REGION Network 13 (SCL): COUNT SELECTED BUTTONS
   IF #settings.current.kp8.buttons <> #settings.old.kp8.buttons THEN
       #count := 0;
       FOR #i := 0 TO #buttonCount DO
           #btnSelected := #settings.current.kp8.buttons[#i].select;
           IF #btnSelected THEN
               #count := #count + 1;
           END_IF;
       END_FOR;
       #btnSlctCount := #count;
   END_IF;
END_REGION

REGION Network 14: SELECT ALL BUTTONS
   #tmrSelAllBtn(IN := #settings.current.kp8.assign.act AND NOT #evalSlct AND (#btnSlctCount < #adjBtnCount),   // TON
                 PT := #ptSelectAll);
   IF #tmrSelAllBtn.Q THEN
       "Select All Buttons"(settings := #settings);
       #evalSlct := TRUE;
   END_IF;
END_REGION

REGION Network 15: DESELECT ALL BUTTONS
   #tmrDeslctAllBtn(IN := #settings.current.kp8.assign.act AND NOT #evalSlct AND (#btnSlctCount = #adjBtnCount),   // TON
                    PT := #ptSelectAll);
   IF #tmrDeslctAllBtn.Q THEN
       "Deselect All Buttons"(settings := #settings);
       #evalSlct := TRUE;
   END_IF;
END_REGION

REGION Network 16: RESET EVAL BUTTON SELECTION
   RUNG wire#powerrail
      I_Contact( #settings.current.kp8.assign.act )
      Contact( #settings.old.kp8.assign.act )
      R_Coil( #evalSlct )
   END_RUNG
   // the same network as SCL:
   IF NOT #settings.current.kp8.assign.act AND #settings.old.kp8.assign.act THEN #evalSlct := FALSE; END_IF;
END_REGION

REGION Network 17: ENTRY TIMEOUT
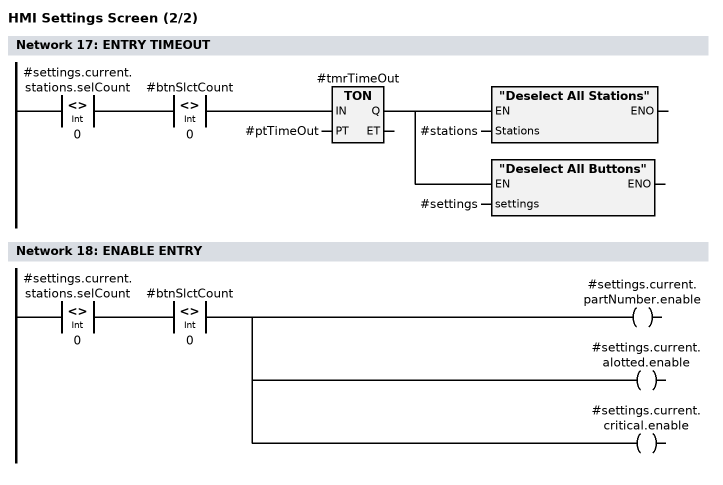
   #tmrTimeOut(IN := (#settings.current.stations.selCount <> 0) AND (#btnSlctCount <> 0), PT := #ptTimeOut);   // TON
   IF #tmrTimeOut.Q THEN
       "Deselect All Stations"(Stations := #stations);
       "Deselect All Buttons"(settings := #settings);
   END_IF;
END_REGION

REGION Network 18: ENABLE ENTRY
   RUNG wire#powerrail
      { S7_Templates := "SrcType := Int" } NE_Contact(in1 := #settings.current.stations.selCount, in2 := 0)
      { S7_Templates := "SrcType := Int" } NE_Contact(in1 := #btnSlctCount, in2 := 0)
      wire#w1
      Coil( #settings.current.partNumber.enable )
   END_RUNG
   RUNG wire#w1
      Coil( #settings.current.alotted.enable )
   END_RUNG
   RUNG wire#w1
      Coil( #settings.current.critical.enable )
   END_RUNG
   // the same network as SCL:
   #settings.current.partNumber.enable := (#settings.current.stations.selCount <> 0) AND (#btnSlctCount <> 0);
   #settings.current.alotted.enable := #settings.current.partNumber.enable;
   #settings.current.critical.enable := #settings.current.partNumber.enable;
END_REGION

REGION Network 19 (SCL): GET BUTTON NUMBER
   IF #btnSlctCount = 1 THEN
       FOR #i := 0 TO #stationCount DO
           #stnSelected := #stations.current[#i].settings.selected;
           IF #stnSelected THEN
               FOR #j := 0 TO #buttonCount DO
                   #btnSelected := #settings.current.kp8.buttons[#j].selState;
                   IF #btnSelected THEN
                       #btnNumber := #j + 1;
                   END_IF;
               END_FOR;
           END_IF;
       END_FOR;
   END_IF;
END_REGION

REGION Network 20 (SCL): DISPLAY PART NUMBER FOR CURRENT BUTTON
   IF #settings.current.viewingStation <> #settings.old.viewingStation THEN
       IF #buttonCount = 1 THEN
           #pSN := #settings.current.viewingStation.number - 1;
           #pBtn := #btnSlctCount - 1;
           #settings.current.partNumber.value := #stations.current[#pSN].partNumbers[#pBtn];
       END_IF;
   END_IF;
END_REGION

REGION Network 21 (SCL): LOAD PART NUMBERS INTO SELECTIONS
   #partNumber := #settings.current.partNumber.value;
   #oldPN := #settings.old.partNumber.value;
   #newEntry := FALSE;
   IF #partNumber <> #oldPN THEN
       #newEntry := TRUE;
   END_IF;
   IF #newEntry THEN
       #newEntry := FALSE;
       FOR #i := 0 TO #constants.stationCount DO
           #stnSelected := #stations.current[#i].settings.selected;
           IF #stnSelected THEN
               FOR #j := 0 TO #constants.buttonCount DO
                   #btnSelected := #settings.current.kp8.buttons[#j].selState;
                   IF #btnSelected THEN
                       #stations.current[#i].partNumbers[#j] := #partNumber;
                   END_IF;
               END_FOR;
           END_IF;
       END_FOR;
   END_IF;
END_REGION

REGION Network 22 (SCL): LOAD TIMER VALUES INTO SELECTIONS
   #currentBtn := #settings.current.alotted.setTimer;
   #oldBtn := #settings.old.alotted.setTimer;
   IF #currentBtn AND NOT #oldBtn THEN
       #timerWString := #settings.current.alotted.value;
       FOR #i := 0 TO #constants.stationCount - 1 DO
           #stnSelected := #stations.current[#i].settings.selected;
           IF #stnSelected THEN
               FOR #j := 0 TO #constants.buttonCount - 1 DO
                   #btnSelected := #settings.current.kp8.buttons[#j].select;
                   IF #btnSelected THEN
                       #stations.current[#i].presetTime.allotted[#j] := "WString Timer to Real"(#timerWString);
                   END_IF;
               END_FOR;
           END_IF;
       END_FOR;
   END_IF;
END_REGION

REGION Network 23 (SCL): LOAD CRITICAL TIME VALUES INTO SELECTIONS
   #currentBtn := #settings.current.critical.setTimer;
   #oldBtn := #settings.old.critical.setTimer;

   IF #currentBtn AND NOT #oldBtn THEN
       #timerWString := #settings.current.alotted.value;
       FOR #i := 0 TO #constants.stationCount - 1 DO
           #stnSelected := #stations.current[#i].settings.selected;
           IF #stnSelected THEN
               FOR #j := 0 TO #constants.buttonCount - 1 DO
                   #btnSelected := #settings.current.kp8.buttons[#j].select;
                   IF #btnSelected THEN
                       #stations.current[#i].presetTime.critical[#j] := "WString Timer to Real"(#timerWString);
                   END_IF;
               END_FOR;
           END_IF;
       END_FOR;
   END_IF;
END_REGION

REGION Network 24 (SCL): UPDATE CURRENT STATION VIEW PORT
   #currentBtn := #settings.current.partNumber.enter OR
                   #settings.current.alotted.setTimer OR
                   #settings.current.critical.setTimer;
   #oldBtn := #settings.old.partNumber.enter OR
                   #settings.old.alotted.setTimer OR
                   #settings.old.critical.setTimer;
   #stnNumber := #settings.current.viewingStation.number;
   #oldStnNumber := #settings.old.viewingStation.number;
   IF (#currentBtn AND NOT #oldBtn) OR
       (#stnNumber <> #oldStnNumber) THEN
       #pSN := #stnNumber - 1;
           // station number: see network 5 & 6
           // line value
           #settings.current.viewingStation.lineValue := #stations.current[#pSN].line;
           // drop zone
           #settings.current.viewingStation.dzValue := #stations.current[#pSN].dropZone;
           // loop through buttons
           FOR #i := 0 TO #constants.buttonCount - 1 DO
               // part number
               #partNumber := #stations.current[#pSN].partNumbers[#i];
               #settings.current.viewingStation.btns[#i].partNumber := #partNumber;
               // allotted time
               #timerWString := "Real to WString Timer"(#stations.current[#pSN].presetTime.allotted[#i]);
               #settings.current.viewingStation.btns[#i].alloted := #timerWString;
               // critical time
               #timerWString := "Real to WString Timer"(#stations.current[#pSN].presetTime.critical[#i]);
               #settings.current.viewingStation.btns[#i].critical := #timerWString;
           END_FOR;
   END_IF;
END_REGION
END_FUNCTION_BLOCK

FUNCTION_BLOCK "Collapse Table"   // FB15, SCL
{ S7_Optimized_Access := 'TRUE' }
VERSION : 0.1
   VAR_INPUT
      constants : "Constants";
   END_VAR
   VAR_IN_OUT
      requests : "Part Request Data";
   END_VAR
   VAR
      tableBox : "Part Request Data";
   END_VAR
   VAR_TEMP
      blankRow : "Table Row";
      collapseReq : Bool;
      i : Int;
      maxRows : Int;
      pCollapse : Int;
   END_VAR
BEGIN
   REGION "COPY TO LOCAL"
       #maxRows := #constants.partReqRows - 1;
   END_REGION

   REGION "REMOVE EMPTY ROWS"
       FOR #i := 0 TO #maxRows DO

           REGION "ROW IS NOT EMPTY"
               IF #requests.row[#i].address <> 0 THEN

                   REGION "MOVE TO TEMP TABLE"
                       #tableBox.row[#pCollapse] := #requests.row[#i];
                   END_REGION

                   REGION "POINTERS AND FLAGS"
                       #pCollapse := #pCollapse + 1;
                       #collapseReq := TRUE;
                   END_REGION

               END_IF;
           END_REGION

       END_FOR;
   END_REGION

   REGION "COLLAPSE TABLE"
       IF #collapseReq THEN

           REGION "TURN OFF THE LIGHTS"
               #collapseReq := FALSE;
           END_REGION

           REGION "COPY TEMP TO PERMANENT"
               #requests := #tableBox;
           END_REGION

           REGION "CLEAR VALUES FROM TEMP TABLE"
               FOR #i := 0 TO #maxRows DO
                   #tableBox.row[#i] := #blankRow;
               END_FOR;
           END_REGION
       END_IF;

   END_REGION
END_FUNCTION_BLOCK

FUNCTION_BLOCK "HMI Populate Part Call"   // FB16, SCL
{ S7_Optimized_Access := 'TRUE' }
VERSION : 0.1
   VAR_INPUT
      constants : "Constants";
      requests : "Part Request Data";
   END_VAR
   VAR_IN_OUT
      partCall : "Part Call Screen";
   END_VAR
   VAR
      pDisplay : Int;
   END_VAR
   VAR_TEMP
      firstRow : Int;
      i : Int;
      lastRow : Int;
      maxRows : Int;
      pRow : Int;
      visibleRows : Int;
      thisRow : Int;
   END_VAR
BEGIN
   #visibleRows := #constants.hmiRowCount - 1;
   #maxRows := #constants.partReqRows - 1;
   #firstRow := 0;
   #lastRow := #firstRow + #visibleRows;

   FOR #i := 0 TO #visibleRows DO
       #partCall.current[#i] := #requests.row[#i];
   END_FOR;
END_FUNCTION_BLOCK

FUNCTION_BLOCK "KP8 Driver"   // FB101, SCL
{ S7_Optimized_Access := 'FALSE' }
VERSION : 0.1
   VAR_INPUT
      btnIn : Byte;   // byte that contains input data from kp8 buttons
      hardInit : Bool;   // initializes function. can be used for reset
      softInit : Bool;
      btn0Activate : Bool;   // true for on, false for off
      btn0Mode : Bool;   // true for maintained, false for momentary
      btn0Group : Int;
      btn0Flash : Bool;
      btn0ColorOn1 : String[10];   // enter: red OR green OR blue OR yellow OR white OR off
      btn0ColorOn2 : String[10];
      btn0ColorOff : String[10];   // enter: red OR green OR blue OR yellow OR white OR off
      btn1Activate : Bool;   // true for on, false for off
      btn1Mode : Bool;   // true for maintained, false for momentary
      btn1Group : Int;
      btn1Flash : Bool;
      btn1ColorOn1 : String[10];   // enter: red OR green OR blue OR yellow OR white OR off
      btn1ColorOn2 : String[10];
      btn1ColorOff : String[10];   // enter: red OR green OR blue OR yellow OR white OR off
      btn2Activate : Bool;   // true for on, false for off
      btn2Mode : Bool;   // true for maintained, false for momentary
      btn2Group : Int;
      btn2Flash : Bool;
      btn2ColorOn1 : String[10] := '';   // enter: red OR green OR blue OR yellow OR white OR off
      btn2ColorOn2 : String[10];
      btn2ColorOff : String[10];   // enter: red OR green OR blue OR yellow OR white OR off
      btn3Activate : Bool;   // true for on, false for off
      btn3Mode : Bool;   // true for maintained, false for momentary
      btn3Group : Int;
      btn3Flash : Bool;
      btn3ColorOn1 : String[10];   // enter: red OR green OR blue OR yellow OR white OR off
      btn3ColorOn2 : String[10];
      btn3ColorOff : String[10];   // enter: red OR green OR blue OR yellow OR white OR off
      btn4Activate : Bool;   // true for on, false for off
      btn4Mode : Bool;   // true for maintained, false for momentary
      btn4Group : Int;
      btn4Flash : Bool;
      btn4ColorOn1 : String[10];   // enter: red OR green OR blue OR yellow OR white OR off
      btn4ColorOn2 : String[10];
      btn4ColorOff : String[10];   // enter: red OR green OR blue OR yellow OR white OR off
      btn5Activate : Bool;   // true for on, false for off
      btn5Mode : Bool;   // true for maintained, false for momentary
      btn5Group : Int;
      btn5Flash : Bool;
      btn5ColorOn1 : String[10];   // enter: red OR green OR blue OR yellow OR white OR off
      btn5ColorOn2 : String[10];
      btn5ColorOff : String[10];   // enter: red OR green OR blue OR yellow OR white OR off
      btn6Activate : Bool;   // true for on, false for off
      btn6Mode : Bool;   // true for maintained, false for momentary
      btn6Group : Int;
      btn6Flash : Bool;
      btn6ColorOn1 : String[10];   // enter: red OR green OR blue OR yellow OR white OR off
      btn6ColorOn2 : String[10];
      btn6ColorOff : String[10];   // enter: red OR green OR blue OR yellow OR white OR off
      btn7Activate : Bool;   // true for on, false for off
      btn7Mode : Bool;   // true for maintained, false for momentary
      btn7Group : Int;
      btn7Flash : Bool;
      btn7ColorOn1 : String[10];   // enter: red OR green OR blue OR yellow OR white OR off
      btn7ColorOn2 : String[10];
      btn7ColorOff : String[10];   // enter: red OR green OR blue OR yellow OR white OR off
   END_VAR
   VAR_OUTPUT
      btnStatesOut : Array[0..7] of Bool;   // the output array represents the state of button presses
      btnColorsOut : DWord;
   END_VAR
   VAR
      mask : Byte;
      btnInInt : Byte;
      btnEval : Byte;
      i1 : Int;
      i2 : Int;
      btnInArrayNew : Array[0..7] of Bool;
      btnInArrayOld : Array[0..7] of Bool;
      btnStateArrayInt : Array[0..7] of Bool;
      btnActivateInt : Array[0..7] of Bool;
      btnModeInt : Array[0..7] of Bool;
      btnFlashInt : Array[0..7] of Bool;
      btnGroup : Array[0..7] of Int;
      btnClrMskOn1Int : Array[0..7] of DWord;
      btnClrMskOn2Int : Array[0..7] of DWord;
      btnClrMskOffInt : Array[0..7] of DWord;
      btnClrOn1Int : Array[0..7] of String[10];
      btnClrOn2Int : Array[0..7] of String[10];
      btnClrOffInt : Array[0..7] of String[10];
   END_VAR
   VAR CONSTANT
      btnMskRed : DWord := dw#16#0100_0000;
      btnMskGreen : DWord := dw#16#0001_0000;
      btnMskBlue : DWord := dw#16#000_0100;
      btnMskYellow : DWord := dw#16#0101_0000;
      btnMskWhite : DWord := dw#16#0101_0100;
      btnMskBlack : DWord := dw#16#FEFE_FEFF;
      initBtnColors : DWord := dw#16#0000_0000;
   END_VAR
BEGIN
   REGION "ALL INITS"
       IF #hardInit OR #softInit THEN

           REGION "CLEAR OUTPUT COLORS"
               #btnColorsOut := #initBtnColors;
           END_REGION

           REGION "TRANSFER PARAMETERS TO INTERNAL ARRAYS"

               REGION "BUTTON 0"
                   #btnActivateInt[0] := #btn0Activate;
                   #btnModeInt[0] := #btn0Mode;
                   #btnGroup[0] := #btn0Group;
                   #btnClrOn1Int[0] := #btn0ColorOn1;
                   #btnClrOn2Int[0] := #btn0ColorOn2;
                   #btnClrOffInt[0] := #btn0ColorOff;
               END_REGION

               REGION "BUTTON 1"
                   #btnActivateInt[1] := #btn1Activate;
                   #btnModeInt[1] := #btn1Mode;
                   #btnGroup[1] := #btn1Group;
                   #btnClrOn1Int[1] := #btn1ColorOn1;
                   #btnClrOn2Int[1] := #btn1ColorOn2;
                   #btnClrOffInt[1] := #btn1ColorOff;
               END_REGION

               REGION "BUTTON 2"
                   #btnActivateInt[2] := #btn2Activate;
                   #btnModeInt[2] := #btn2Mode;
                   #btnGroup[2] := #btn2Group;
                   #btnClrOn1Int[2] := #btn2ColorOn1;
                   #btnClrOn2Int[2] := #btn2ColorOn2;
                   #btnClrOffInt[2] := #btn2ColorOff;
               END_REGION

               REGION "BUTTON 3"
                   #btnActivateInt[3] := #btn3Activate;
                   #btnModeInt[3] := #btn3Mode;
                   #btnGroup[3] := #btn3Group;
                   #btnClrOn1Int[3] := #btn3ColorOn1;
                   #btnClrOn2Int[3] := #btn3ColorOn2;
                   #btnClrOffInt[3] := #btn3ColorOff;
               END_REGION

               REGION "BUTTON 4"
                   #btnActivateInt[4] := #btn4Activate;
                   #btnModeInt[4] := #btn4Mode;
                   #btnGroup[4] := #btn4Group;
                   #btnClrOn1Int[4] := #btn4ColorOn1;
                   #btnClrOn2Int[4] := #btn4ColorOn2;
                   #btnClrOffInt[4] := #btn4ColorOff;
               END_REGION

               REGION "BUTTON 5"
                   #btnActivateInt[5] := #btn5Activate;
                   #btnModeInt[5] := #btn5Mode;
                   #btnGroup[5] := #btn5Group;
                   #btnClrOn1Int[5] := #btn5ColorOn1;
                   #btnClrOn2Int[5] := #btn5ColorOn2;
                   #btnClrOffInt[5] := #btn5ColorOff;
               END_REGION

               REGION "BUTTON 6"
                   #btnActivateInt[6] := #btn6Activate;
                   #btnModeInt[6] := #btn6Mode;
                   #btnGroup[6] := #btn6Group;
                   #btnClrOn1Int[6] := #btn6ColorOn1;
                   #btnClrOn2Int[6] := #btn6ColorOn2;
                   #btnClrOffInt[6] := #btn6ColorOff;
               END_REGION

               REGION "BUTTON 7"
                   #btnActivateInt[7] := #btn7Activate;
                   #btnModeInt[7] := #btn7Mode;
                   #btnGroup[7] := #btn7Group;
                   #btnClrOn1Int[7] := #btn7ColorOn1;
                   #btnClrOn2Int[7] := #btn7ColorOn2;
                   #btnClrOffInt[7] := #btn7ColorOff;
               END_REGION

           END_REGION

           REGION "RECOLOR BUTTON MASKS"
               FOR #i1 := 0 TO 7 DO

                   REGION "ON COLOR 1"
                       IF (#btnClrOn1Int[#i1] = 'red') THEN
                           #btnClrMskOn1Int[#i1] := SHL(IN := #btnMskRed, N := #i1);
                       ELSIF (#btnClrOn1Int[#i1] = 'green') THEN
                           #btnClrMskOn1Int[#i1] := SHL(IN := #btnMskGreen, N := #i1);
                       ELSIF (#btnClrOn1Int[#i1] = 'blue') THEN
                           #btnClrMskOn1Int[#i1] := SHL(IN := #btnMskBlue, N := #i1);
                       ELSIF (#btnClrOn1Int[#i1] = 'yellow') THEN
                           #btnClrMskOn1Int[#i1] := SHL(IN := #btnMskYellow, N := #i1);
                       ELSIF (#btnClrOn1Int[#i1] = 'white') THEN
                           #btnClrMskOn1Int[#i1] := SHL(IN := #btnMskWhite, N := #i1);
                       ELSIF (#btnClrOn1Int[#i1] = 'off') THEN
                           #btnClrMskOn1Int[#i1] := 0;
                       END_IF;
                   END_REGION

                   REGION "ON COLOR 2"
                       IF (#btnClrOn2Int[#i1] = 'red') THEN
                           #btnClrMskOn2Int[#i1] := SHL(IN := #btnMskRed, N := #i1);
                       ELSIF (#btnClrOn2Int[#i1] = 'green') THEN
                           #btnClrMskOn2Int[#i1] := SHL(IN := #btnMskGreen, N := #i1);
                       ELSIF (#btnClrOn2Int[#i1] = 'blue') THEN
                           #btnClrMskOn2Int[#i1] := SHL(IN := #btnMskBlue, N := #i1);
                       ELSIF (#btnClrOn2Int[#i1] = 'yellow') THEN
                           #btnClrMskOn2Int[#i1] := SHL(IN := #btnMskYellow, N := #i1);
                       ELSIF (#btnClrOn2Int[#i1] = 'white') THEN
                           #btnClrMskOn2Int[#i1] := SHL(IN := #btnMskWhite, N := #i1);
                       ELSIF (#btnClrOn2Int[#i1] = 'off') THEN
                           #btnClrMskOn2Int[#i1] := 0;
                       END_IF;
                   END_REGION

                   REGION "OFF COLOR"
                       IF (#btnClrOffInt[#i1] = 'red') THEN
                           #btnClrMskOffInt[#i1] := SHL(IN := #btnMskRed, N := #i1);
                       ELSIF (#btnClrOffInt[#i1] = 'green') THEN
                           #btnClrMskOffInt[#i1] := SHL(IN := #btnMskGreen, N := #i1);
                       ELSIF (#btnClrOffInt[#i1] = 'blue') THEN
                           #btnClrMskOffInt[#i1] := SHL(IN := #btnMskBlue, N := #i1);
                       ELSIF (#btnClrOffInt[#i1] = 'yellow') THEN
                           #btnClrMskOffInt[#i1] := SHL(IN := #btnMskYellow, N := #i1);
                       ELSIF (#btnClrOffInt[#i1] = 'white') THEN
                           #btnClrMskOffInt[#i1] := SHL(IN := #btnMskWhite, N := #i1);
                       ELSIF (#btnClrOffInt[#i1] = 'off') THEN
                           #btnClrMskOffInt[#i1] := 0;
                       END_IF;
                   END_REGION

               END_FOR;
           END_REGION

       END_IF;
   END_REGION

   REGION "HART INIT"
       IF #hardInit THEN
           FOR #i1 := 0 TO 7 DO
               #btnStateArrayInt[#i1] := FALSE;
           END_FOR;
       END_IF;
   END_REGION


   REGION "TRANFER PARAMETERS TO ARRAYS"
       // raw pb data
       #btnInInt := #btnIn;
       // flashing modes
       #btnFlashInt[0] := #btn0Flash;
       #btnFlashInt[1] := #btn1Flash;
       #btnFlashInt[2] := #btn2Flash;
       #btnFlashInt[3] := #btn3Flash;
       #btnFlashInt[4] := #btn4Flash;
       #btnFlashInt[5] := #btn5Flash;
       #btnFlashInt[6] := #btn6Flash;
       #btnFlashInt[7] := #btn7Flash;
   END_REGION

   REGION "EVALUATE BUTTONS"
       FOR #i1 := 0 TO 7 DO

           REGION "TRANSFER BUTTON PRESSES TO ARRAY"
               #btnEval := SHR(IN := #btnInInt, N := #i1);
               #btnInArrayNew[#i1] := #btnEval.%X0;
               #btnEval := b#16#0;
           END_REGION

           REGION "SET BUTTON STATE"

               REGION "BUTTON ACTIVE"
                   IF #btnActivateInt[#i1] THEN

                       REGION "MAINTAINED"
                           IF #btnModeInt[#i1] THEN

                               REGION "RISING EDGE OF PRESS"
                                   IF #btnInArrayNew[#i1] AND NOT #btnInArrayOld[#i1] THEN

                                       REGION "CHECK FOR GROUP MEMBERSHIP"
                                           FOR #i2 := 0 TO 7 DO

                                               REGION "NOT IN NULL GROUP"
                                                   IF (#btnGroup[#i2] <> 0) THEN

                                                       REGION "SKIP SELF"
                                                           IF (#i2 <> #i1) THEN

                                                               REGION "GROUPS MATCH"
                                                                   IF #btnGroup[#i1] = #btnGroup[#i2] THEN
                                                                       REGION "DEACTIVATE OTHER GROUP MEMBERS"
                                                                           #btnStateArrayInt[#i2] := FALSE;
                                                                       END_REGION

                                                                   END_IF;
                                                               END_REGION

                                                           END_IF;
                                                       END_REGION

                                                   END_IF;
                                               END_REGION

                                           END_FOR;
                                       END_REGION

                                       REGION "TOGGLE STATE"
                                           #btnStateArrayInt[#i1] := NOT #btnStateArrayInt[#i1];
                                       END_REGION

                                   END_IF;
                               END_REGION

                           END_IF;
                       END_REGION

                       REGION "MOMENTARY"
                           IF NOT #btnModeInt[#i1] THEN
                               #btnStateArrayInt[#i1] := #btnInArrayNew[#i1];
                           END_IF;
                       END_REGION

                   END_IF;
               END_REGION

               REGION "BUTTON INACTIVE"
                   IF NOT #btnActivateInt[#i1] THEN
                       #btnStateArrayInt[#i1] := FALSE;
                   END_IF;
               END_REGION

           END_REGION

           REGION "ANIMATE BUTTONS"

               REGION "BUTTON ON FLASH BIT OFF"
                   IF #btnStateArrayInt[#i1] AND NOT #btnFlashInt[#i1] THEN
                       #btnColorsOut := #btnColorsOut AND ROL(IN := #btnMskBlack, N := #i1);
                       #btnColorsOut := #btnColorsOut OR #btnClrMskOn1Int[#i1];
                   END_IF;
               END_REGION

               REGION "BUTTON ON FLASH BIT ON"
                   IF #btnStateArrayInt[#i1] AND #btnFlashInt[#i1] THEN
                       #btnColorsOut := #btnColorsOut AND ROL(IN := #btnMskBlack, N := #i1);
                       #btnColorsOut := #btnColorsOut OR #btnClrMskOn2Int[#i1];
                   END_IF;
               END_REGION

               REGION "BUTTON OFF"
                   IF NOT #btnStateArrayInt[#i1] THEN
                       #btnColorsOut := #btnColorsOut AND ROL(IN := #btnMskBlack, N := #i1);
                       #btnColorsOut := #btnColorsOut OR #btnClrMskOffInt[#i1];
                   END_IF;
               END_REGION

           END_REGION

       END_FOR;
   END_REGION

   REGION "CHANGE DETECTION"
       #btnInArrayOld := #btnInArrayNew;
   END_REGION

   REGION "OUTPUT"
       #btnStatesOut := #btnStateArrayInt;
   END_REGION
END_FUNCTION_BLOCK

FUNCTION "Physical to Global" : Void   // FC1, LAD
{ S7_Optimized_Access := 'TRUE' }
VERSION : 0.1
   VAR_INPUT
      constants : "Constants";
   END_VAR
   VAR_IN_OUT
      stations : "Stations";
   END_VAR
   VAR_TEMP
      i : Int;
      kp8In : DWord;
      stnCount : Int;
   END_VAR
   VAR CONSTANT
      "VOLVO 16 1" : Int := 0;
      "VOLVO 16 2" : Int := 1;
      "VOLVO 16 3" : Int := 2;
      "VOLVO 16 4" : Int := 3;
      "VOLVO 16 5" : Int := 4;
      "VOLVO 16 6" : Int := 5;
      "VOLVO 16 7" : Int := 6;
      "VOLVO 16 8" : Int := 7;
      "VOLVO 16 9" : Int := 8;
      "VOLVO 16 10" : Int := 9;
      "VOLVO 16 11" : Int := 10;
      "CHM 1" : Int := 11;
      "CHM 2" : Int := 12;
      "CHM 3" : Int := 13;
      "CHM 4" : Int := 14;
      "CDO 1" : Int := 15;
      "CDO 2" : Int := 16;
      "CDO 3" : Int := 17;
      "BFL 1" : Int := 18;
      "BFL 2" : Int := 19;
      "BFL 3" : Int := 20;
      "LGS 1" : Int := 21;
      "LGS 2" : Int := 22;
   END_VAR
BEGIN

REGION Network 1
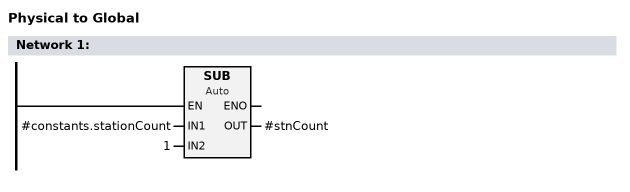
   RUNG wire#powerrail
      Sub(in1 := #constants.stationCount, in2 := 1, out => #stnCount)
   END_RUNG
   // the same network as SCL:
   #stnCount := #constants.stationCount - 1;
END_REGION

REGION Network 2 (SCL): MAIN LOOP
   FOR #i := 0 TO #stnCount DO

       CASE #i OF
           #"VOLVO 16 1":
               #kp8In := "VOLVO 16 1 KP8 In";
           #"VOLVO 16 2":
               #kp8In := "VOLVO 16 2 KP8 In";
           #"VOLVO 16 3":
               #kp8In := "VOLVO 16 3 KP8 In";
           #"VOLVO 16 4":
               #kp8In := "VOLVO 16 4 KP8 In";
           #"VOLVO 16 5":
               #kp8In := "VOLVO 16 5 KP8 In";
           #"VOLVO 16 6":
               #kp8In := "VOLVO 16 6 KP8 In";
           #"VOLVO 16 7":
               #kp8In := "VOLVO 16 7 KP8 In";
           #"VOLVO 16 8":
               #kp8In := "VOLVO 16 8 KP8 In";
           #"VOLVO 16 9":
               #kp8In := "VOLVO 16 9 KP8 In";
           #"VOLVO 16 10":
               #kp8In := "VOLVO 16 10 KP8 In";
           #"VOLVO 16 11":
               #kp8In := "VOLVO 16 11 KP8 In";
           #"CHM 1":
               #kp8In := "CHM 1 KP8 In";
           #"CHM 2":
               #kp8In := "CHM 2 KP8 In";
           #"CHM 3":
               #kp8In := "CHM 3 KP8 In";
           #"CHM 4":
               #kp8In := "CHM 4 KP8 In";
           #"CDO 1":
               #kp8In := "CDO 1 KP8 In";
           #"CDO 2":
               #kp8In := "CDO 2 KP8 In";
           #"CDO 3":
               #kp8In := "CDO 3 KP8 In";
           #"BFL 1":
               #kp8In := "BFL 1 KP8 In";
           #"BFL 2":
               #kp8In := "BFL 2 KP8 In";
           #"BFL 3":
               #kp8In := "BFL 3 KP8 In";
           #"LGS 1":
               #kp8In := "LGS 1 KP8 In";
           #"LGS 2":
               #kp8In := "LGS 2 KP8 In";

       END_CASE;

       #stations.current[#i].kp8In := #kp8In.%B3;

   END_FOR;
END_REGION
END_FUNCTION

FUNCTION "Time to WString" : WString   // FC2, SCL
{ S7_Optimized_Access := 'TRUE' }
VERSION : 0.1
   VAR_INPUT
      "Time" : Time;
   END_VAR
   VAR_TEMP
      "Time as DInt" : DInt;
      "Hours 10s Place" : DInt;
      "Hours 1s Place" : DInt;
      "Minutes 10s Place" : DInt;
      "Minutes 1s Place" : DInt;
      "Seconds 10s Place" : DInt;
      "Seconds 1s Place" : DInt;
      "Time Elements" : Array[0..4] of WString;
      Length : Int;
      "String Box" : WString;
      "DInt Box" : DInt;
   END_VAR
   VAR CONSTANT
      "Milliseconds per 10 Hours" : DInt := 36000000;
      "Milliseconds per Hour" : DInt := 3600000;
      "Milliseconds per 10 Minutes" : DInt := 600000;
      "Milliseconds per Minute" : DInt := 60000;
      "Milliseconds per 10 Seconds" : DInt := 10000;
      "Milliseconds per Second" : DInt := 1000;
   END_VAR
BEGIN
   REGION GET INPUT
       #"Time as DInt" := #Time;
   END_REGION

   REGION CONVERT TIME INTO INDIVIDUAL PLACE VALUES
       #"Minutes 10s Place" := #"Time as DInt" / #"Milliseconds per 10 Minutes";
       #"Minutes 1s Place" := (#"Time as DInt" / #"Milliseconds per Minute") MOD 10;
       #"Seconds 10s Place" := (#"Time as DInt" MOD #"Milliseconds per Minute") / #"Milliseconds per 10 Seconds";
       #"Seconds 1s Place" := (#"Time as DInt" / #"Milliseconds per Second") MOD 10;
   END_REGION

   REGION "ADD SIGN"
       #"Time Elements"[0] := wstring#'';
       IF #"Minutes 10s Place" < 0 OR
           #"Minutes 1s Place" < 0 OR
           #"Seconds 10s Place" < 0 OR
           #"Seconds 1s Place" < 0 THEN
            #"Time Elements"[0] := wstring#'-';
       END_IF;
   END_REGION

   REGION CONVERT PLACE VALUES INTO COMPONENT STRINGS
       // MINUTES
       #"DInt Box" := #"Minutes 10s Place" * 10 + #"Minutes 1s Place";
       #"String Box" := DINT_TO_WSTRING(IN := #"DInt Box");
       #"String Box" := "Strip Sign"("WString":=#"String Box");
       #"String Box" := "Add Leading"("Leading Character" := WCHAR#'0',
                                      "Desired Length" := 2,
                                      "String" := #"String Box");
       #"Time Elements"[1] := #"String Box";
       // COLON
       #"Time Elements"[2] := WSTRING#':';
       // SECONDS
       #"DInt Box" := #"Seconds 10s Place" * 10 + #"Seconds 1s Place";
       #"String Box" := DINT_TO_WSTRING(IN := #"DInt Box");
       #"String Box" := "Strip Sign"("WString":=#"String Box");
       #"String Box" := "Add Leading"("Leading Character" := WCHAR#'0',
                                      "Desired Length" := 2,
                                      "String" := #"String Box");
       #"Time Elements"[3] := #"String Box";
   END_REGION


   REGION RETURN VALUE
       #"Time to WString" := CONCAT_WSTRING(IN1 := #"Time Elements"[0],
                                            IN2 := #"Time Elements"[1],
                                            IN3 := #"Time Elements"[2],
                                            IN4 := #"Time Elements"[3]);
   END_REGION
END_FUNCTION

FUNCTION "Strip Sign" : WString   // FC3, SCL
{ S7_Optimized_Access := 'TRUE' }
VERSION : 0.1
   VAR_INPUT
      WString : WString;
   END_VAR
   VAR_TEMP
      Length : Int;
      "String Box" : WString;
      "Test Character" : WString;
   END_VAR
   VAR CONSTANT
      "+" : WChar := WCHAR#'+';
      "-" : WChar := WCHAR#'-';
   END_VAR
BEGIN
   #"String Box" := #WString;
   #"Test Character" := LEFT_WSTRING(IN := #"String Box",
                                     L := 1);
   IF #"Test Character" = #"+" OR #"Test Character" = #"-" THEN
       #Length := LEN(#"String Box");
       #"String Box" := RIGHT_WSTRING(IN := #"String Box", L := #Length - 1);

   END_IF;
   #"Strip Sign" := #"String Box";
END_FUNCTION

FUNCTION "Add Leading" : WString   // FC4, SCL
{ S7_Optimized_Access := 'TRUE' }
VERSION : 0.1
   VAR_INPUT
      "Leading Character" : WChar;
      "Desired Length" : USInt;
      "String" : WString;
   END_VAR
   VAR_TEMP
      Length : Int;
      "String Box" : WString;
      Constant : WString;
   END_VAR
BEGIN
   #"String Box" := #String;
   #Length := LEN(#"String Box");

   WHILE #Length < #"Desired Length" DO
       #"String Box" := CONCAT_WSTRING(IN1 := #"Leading Character",
                                       IN2 := #"String Box");
       #Length := LEN(#"String Box");
   END_WHILE;

   #"Add Leading" := #"String Box";
END_FUNCTION

FUNCTION "Global to Physical" : Void   // FC5, LAD
{ S7_Optimized_Access := 'TRUE' }
VERSION : 0.1
   VAR_INPUT
      constants : "Constants";
   END_VAR
   VAR_IN_OUT
      stations : "Stations";
   END_VAR
   VAR_TEMP
      i : Int;
      j : Int;
      IO : DWord;
      "KP8 In" : DWord;
      "KP8 Out" : DWord;
      Card : Int;
      stnCount : Int;
   END_VAR
   VAR CONSTANT
      "VOLVO 16 1" : Int := 0;
      "VOLVO 16 2" : Int := 1;
      "VOLVO 16 3" : Int := 2;
      "VOLVO 16 4" : Int := 3;
      "VOLVO 16 5" : Int := 4;
      "VOLVO 16 6" : Int := 5;
      "VOLVO 16 7" : Int := 6;
      "VOLVO 16 8" : Int := 7;
      "VOLVO 16 9" : Int := 8;
      "VOLVO 16 10" : Int := 9;
      "VOLVO 16 11" : Int := 10;
      "CHM 1" : Int := 11;
      "CHM 2" : Int := 12;
      "CHM 3" : Int := 13;
      "CHM 4" : Int := 14;
      "CDO 1" : Int := 15;
      "CDO 2" : Int := 16;
      "CDO 3" : Int := 17;
      "BFL 1" : Int := 18;
      "BFL 2" : Int := 19;
      "BFL 3" : Int := 20;
      "LGS 1" : Int := 21;
      "LGS 2" : Int := 22;
   END_VAR
BEGIN

REGION Network 1: ARRAY LIMIT FOR STATION COUNT
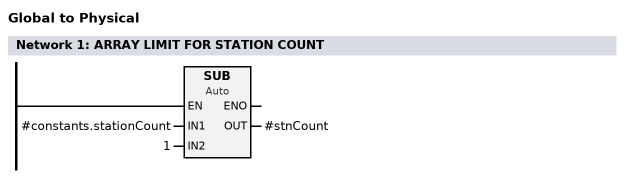
   RUNG wire#powerrail
      Sub(in1 := #constants.stationCount, in2 := 1, out => #stnCount)
   END_RUNG
   // the same network as SCL:
   #stnCount := #constants.stationCount - 1;
END_REGION

REGION Network 2 (SCL): MAIN LOOP
   FOR #i := 0 TO #stnCount DO

       #IO := #stations.current[#i].stackLightOut;
       #"KP8 Out" := #stations.current[#i].kp8Out;

       CASE #i OF
           #"VOLVO 16 1":
               "VOLVO 16 1 IO" := #IO;
               "VOLVO 16 1 KP8 Out" := #"KP8 Out";
           #"VOLVO 16 2":
               "VOLVO 16 2 IO" := #IO;
               "VOLVO 16 2 KP8 Out" := #"KP8 Out";
           #"VOLVO 16 3":
               "VOLVO 16 3 IO" := #IO;
               "VOLVO 16 3 KP8 Out" := #"KP8 Out";
           #"VOLVO 16 4":
               "VOLVO 16 4 IO" := #IO;
               "VOLVO 16 4 KP8 Out" := #"KP8 Out";
           #"VOLVO 16 5":
               "VOLVO 16 5 IO" := #IO;
               "VOLVO 16 5 KP8 Out" := #"KP8 Out";
           #"VOLVO 16 6":
               "VOLVO 16 6 IO" := #IO;
               "VOLVO 16 6 KP8 Out" := #"KP8 Out";
           #"VOLVO 16 7":
               "VOLVO 16 7 IO" := #IO;
               "VOLVO 16 7 KP8 Out" := #"KP8 Out";
           #"VOLVO 16 8":
               "VOLVO 16 8 IO" := #IO;
               "VOLVO 16 8 KP8 Out" := #"KP8 Out";
           #"VOLVO 16 9":
               "VOLVO 16 9 IO" := #IO;
               "VOLVO 16 9 KP8 Out" := #"KP8 Out";
           #"VOLVO 16 10":
               "VOLVO 16 10 IO" := #IO;
               "VOLVO 16 10 KP8 Out" := #"KP8 Out";
           #"VOLVO 16 11":
               "VOLVO 16 11 IO" := #IO;
               "VOLVO 16 11 KP8 Out" := #"KP8 Out";
           #"CHM 1":
               "CHM 1 IO" := #IO;
               "CHM 1 KP8 Out" := #"KP8 Out";
           #"CHM 2":
               "CHM 2 IO" := #IO;
               "CHM 2 KP8 Out" := #"KP8 Out";
           #"CHM 3":
               "CHM 3 IO" := #IO;
               "CHM 3 KP8 Out" := #"KP8 Out";
           #"CHM 4":
               "CHM 4 IO" := #IO;
               "CHM 4 KP8 Out" := #"KP8 Out";
           #"CDO 1":
               "CDO 1 IO" := #IO;
               "CDO 1 KP8 Out" := #"KP8 Out";
           #"CDO 2":
               "CDO 2 IO" := #IO;
               "CDO 2 KP8 Out" := #"KP8 Out";
           #"CDO 3":
               "CDO 3 IO" := #IO;
               "CDO 3 KP8 Out" := #"KP8 Out";
           #"BFL 1":
               "BFL 1 IO" := #IO;
               "BFL 1 KP8 Out" := #"KP8 Out";
           #"BFL 2":
               "BFL 2 IO" := #IO;
               "BFL 2 KP8 Out" := #"KP8 Out";
           #"BFL 3":
               "BFL 3 IO" := #IO;
               "BFL 3 KP8 Out" := #"KP8 Out";
           #"LGS 1":
               "LGS 1 IO" := #IO;
               "LGS 1 KP8 Out" := #"KP8 Out";
           #"LGS 2":
               "LGS 2 IO" := #IO;
               "LGS 2 KP8 Out" := #"KP8 Out";

       END_CASE;

   END_FOR;
END_REGION
END_FUNCTION

FUNCTION "Select All Stations" : Void   // FC6, SCL
{ S7_Optimized_Access := 'TRUE' }
VERSION : 0.1
   VAR_IN_OUT
      stations : "Stations";
   END_VAR
   VAR_TEMP
      i : Int;
   END_VAR
   VAR CONSTANT
      stationCount : Int := 22;
   END_VAR
BEGIN
   FOR #i := 0 TO #stationCount DO 
       #stations.current[#i].settings.selected := TRUE;
   END_FOR;
END_FUNCTION

FUNCTION "Deselect All Stations" : Void   // FC7, SCL
{ S7_Optimized_Access := 'TRUE' }
VERSION : 0.1
   VAR_IN_OUT
      Stations : "Stations";
   END_VAR
   VAR_TEMP
      i : Int;
   END_VAR
   VAR CONSTANT
      stationCount : Int := 10;
   END_VAR
BEGIN
   FOR #i := 0 TO #stationCount DO
       #Stations.current[#i].settings.selected := FALSE;
   END_FOR;
END_FUNCTION

FUNCTION "Select All Buttons" : Void   // FC8, SCL
{ S7_Optimized_Access := 'TRUE' }
VERSION : 0.1
   VAR_IN_OUT
      settings : "Settings Screen";
   END_VAR
   VAR_TEMP
      i : Int;
   END_VAR
   VAR CONSTANT
      buttonCount : Int := 5;
   END_VAR
BEGIN
   FOR #i := 0 TO #buttonCount DO 
       #settings.current.kp8.buttons[#i].select := TRUE;
   END_FOR;
END_FUNCTION

FUNCTION "Deselect All Buttons" : Void   // FC9, SCL
{ S7_Optimized_Access := 'TRUE' }
VERSION : 0.1
   VAR_IN_OUT
      settings : "Settings Screen";
   END_VAR
   VAR_TEMP
      i : Int;
   END_VAR
   VAR CONSTANT
      buttonCount : Int := 5;
   END_VAR
BEGIN
   FOR #i := 0 TO #buttonCount DO
       #settings.current.kp8.buttons[#i].select := FALSE;
   END_FOR;
END_FUNCTION

FUNCTION "WString to Time" : Time   // FC10, SCL
{ S7_Optimized_Access := 'TRUE' }
VERSION : 0.1
   VAR_INPUT
      WString : WString;
   END_VAR
   VAR_TEMP
      Count : UInt;
      "DInt Box" : DInt;
      "String Box" : WString [5];
      "Time Box" : Time;
      "WChar Array" : Array[0..4] of WChar;
   END_VAR
   VAR CONSTANT
      "ms/(10 hr)" : DInt := 36000000;
      "ms/hr" : DInt := 3600000;
      "ms/(10 min)" : DInt := 600000;
      "ms/min" : DInt := 60000;
      "ms/(10 sec)" : DInt := 10000;
      "ms/sec" : DInt := 1000;
   END_VAR
BEGIN
   REGION EXPLODE INPUT

       #"String Box" := #WString;
       IF #"String Box" = WSTRING#'' THEN
           #"String Box" := WSTRING#'00:00';
       END_IF;

       Strg_TO_Chars(Strg := #"String Box",
                     pChars := 0,
                     Cnt => #Count,
                     Chars := #"WChar Array");

   END_REGION

   REGION CONVERT ARRAY ELEMENTS TO TIME

       // 10S OF MINUTES
       #"DInt Box" := WCHAR_TO_DINT(IN := #"WChar Array"[0]) - 16#30;
       #"Time Box" := #"Time Box" + #"DInt Box" * #"ms/(10 min)";

       // MINUTES
       #"DInt Box" := WCHAR_TO_DINT(IN := #"WChar Array"[1]) - 16#30;
       #"Time Box" := #"Time Box" + #"DInt Box" * #"ms/min";

       // 10S OF SECONDS
       #"DInt Box" := WCHAR_TO_DINT(IN := #"WChar Array"[3]) - 16#30;
       #"Time Box" := #"Time Box" + #"DInt Box" * #"ms/(10 sec)";

       // SECONDS
       #"DInt Box" := WCHAR_TO_DINT(IN := #"WChar Array"[4]) - 16#30;
       #"Time Box" := #"Time Box" + #"DInt Box" * #"ms/sec";

   END_REGION


   REGION RETURN VALUE

       #"WString to Time" := #"Time Box";

   END_REGION
END_FUNCTION

FUNCTION "Get Part Call Row Number" : Int   // FC11, SCL
{ S7_Optimized_Access := 'TRUE' }
VERSION : 0.1
   VAR_INPUT
      constants : "Constants";
   END_VAR
   VAR_IN_OUT
      partCall : "Part Call Screen";
   END_VAR
   VAR_TEMP
      hmiRows : Int;
      i : Int;
      selectedRow : Int;
   END_VAR
BEGIN
   REGION "GET NUMBER OF HMI ROWS"
       #hmiRows := #constants.hmiRowCount - 1;
   END_REGION

   REGION "LOOP THROUGH HMI ROWS
       FOR #i := 0 TO #hmiRows DO

           REGION "FIND SELECTED ROW"
               IF #partCall.current[#i].pbSelection.request THEN
                   // turn off the lights
                   #partCall.current[#i].pbSelection.request := FALSE;
                   // selected row as int
                   #selectedRow := #i + 1;
                   EXIT;
               END_IF;
           END_REGION

       END_FOR;
   END_REGION

   REGION "RETURN ROW NUMBER"
       #"Get Part Call Row Number" := #selectedRow;
   END_REGION
END_FUNCTION

FUNCTION "Address to Station and Button" : Void   // FC12, SCL
{ S7_Optimized_Access := 'TRUE' }
VERSION : 0.1
   VAR_INPUT
      address : UInt;
   END_VAR
   VAR_OUTPUT
      station : UInt;
      button : UInt;
   END_VAR
BEGIN
   #station := #address / 10;
   #button := #address MOD 10;
END_FUNCTION

FUNCTION "WString Timer to Real" : Real   // FC13, SCL
{ S7_Optimized_Access := 'TRUE' }
VERSION : 0.1
   VAR_INPUT
      wstring : WString;
   END_VAR
   VAR CONSTANT
      msPerSec : Real := 1000.0;
   END_VAR
BEGIN
   #"WString Timer to Real" := DINT_TO_REAL(TIME_TO_DINT("WString to Time"(#wstring))) / #msPerSec;
END_FUNCTION

FUNCTION "Real to WString Timer" : WString   // FC14, SCL
{ S7_Optimized_Access := 'TRUE' }
VERSION : 0.1
   VAR_INPUT
      realVal : Real;
   END_VAR
   VAR CONSTANT
      msPerSec : Real := 1000.0;
   END_VAR
BEGIN
   #"Real to WString Timer" := "Time to WString"(DINT_TO_TIME(REAL_TO_DINT(#realVal * #msPerSec)));
END_FUNCTION

ORGANIZATION_BLOCK "Main"   // OB1, LAD, ProgramCycle
TITLE = "Main Program Sweep (Cycle)"
{ S7_Optimized_Access := 'TRUE' }
VERSION : 0.1
   VAR_INPUT
      Initial_Call : Bool;   // Initial call of this OB
      Remanence : Bool;   // =True, if remanent data are available
   END_VAR
BEGIN

REGION Network 1
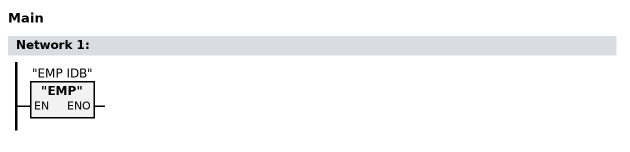
   RUNG wire#powerrail
      "EMP IDB"()
   END_RUNG
   // the same network as SCL:
   "EMP IDB"();   // "EMP"
END_REGION
END_ORGANIZATION_BLOCK

ORGANIZATION_BLOCK "Rack or station failure"   // OB86, LAD, RackStationFailure
{ S7_Optimized_Access := 'TRUE' }
VERSION : 0.1
   VAR_INPUT
      LADDR : Hw_Device;   // Hardware identifier
      Event_Class : Byte;   // Event class
      Fault_ID : Byte;   // Fault identifier
   END_VAR
BEGIN
END_ORGANIZATION_BLOCK

ORGANIZATION_BLOCK "IO access error"   // OB122, LAD, IOAccessError
{ S7_Optimized_Access := 'TRUE' }
VERSION : 0.1
   VAR_INPUT
      BlockNr : UInt;   // Number of causing block
      Reaction : USInt;   // 0:ignore, 1:substitute, 2:skip
      Fault_ID : Byte;   // 16#42:reading, 16#43:writing
      BlockType : USInt;   // 16#01:OB, 16#02:FC, 16#03:FB, 16#04:SFC, 16#05:SFB, 16#06:DB: Type of block causing the error
      Area : USInt;   // 16#81:I, 16#82:Q: IO area where the IOaccess error occured
      DBNr : DB_ANY;   // Reserved for system
      Csg_OBNr : OB_Any;   // Number of OB causing the error
      Csg_Prio : USInt;   // Priority of OB causing the error
      Width : USInt;   // 0:bit, 1:byte, 2:word, 3:dword, 4:lword
   END_VAR
BEGIN
END_ORGANIZATION_BLOCK

// ===== library types =====

TYPE "Table Row Data"
   STRUCT
      address : UInt;
      ordered : Bool;
      pbSelection : Struct
         request : Bool;
         visibility : Bool;
      END_STRUCT;
      rtBackground : Struct
         animatior : UInt;
         visibility : Bool;
      END_STRUCT;
      selected : Bool;
      tfDropZone : Struct
         value : WString[20];
         animator : UInt;
         visibility : Bool;
      END_STRUCT;
      tfLine : Struct
         value : WString[20];
         animator : UInt;
         visibility : Bool;
      END_STRUCT;
      tfPartNumber : Struct
         value : WString[40];
         animator : UInt;
         visibility : Bool;
      END_STRUCT;
      tfTime : Struct
         value : WString[20];
         animator : UInt;
         visibility : Bool;
      END_STRUCT;
   END_STRUCT;
END_TYPE

(* ===== HMI "HMI_RT_1" =====
system functions are stored by id; their names below are inferred from use
connection "HMI_Connection_2": ETHERNET, S7_1500_OMS

HMI tags "Default tag table"
   "Clock_Byte" : Byte = PLC Clock_Byte AT %MB0, 100 ms
   "HMI_screenNumber" : Int = PLC HMI.screenNumber AT %DB1.DBW0, 100 ms
   "HMI_partCall" : Part Call Screen = PLC HMI.partCall AT %DB1.DBW0, 100 ms
   "HMI_settings" : Settings Screen = PLC HMI.settings AT %DB1.DBW0, 100 ms
   "HMI_barcode" : Barcode Screen = PLC HMI.barcode AT %DB1.DBW0, 100 ms
   "HMI_partCall_current{0}" : Table Row = PLC HMI.partCall.current[0], 100 ms
   "HMI_partCall_current{1}" : Table Row = PLC HMI.partCall.current[1], 100 ms
   "HMI_partCall_current{2}" : Table Row = PLC HMI.partCall.current[2], 100 ms
   "HMI_partCall_current{3}" : Table Row = PLC HMI.partCall.current[3], 100 ms
   "HMI_partCall_current{4}" : Table Row = PLC HMI.partCall.current[4], 100 ms
   "HMI_partCall_current{5}" : Table Row = PLC HMI.partCall.current[5], 100 ms
   "HMI_partCall_current{6}" : Table Row = PLC HMI.partCall.current[6], 100 ms
   "HMI_partCall_current{7}" : Table Row = PLC HMI.partCall.current[7], 100 ms
   "HMI_partCall_current{8}" : Table Row = PLC HMI.partCall.current[8], 100 ms
   "HMI_partCall_current{9}" : Table Row = PLC HMI.partCall.current[9], 100 ms
   "HMI_partCall_current{10}" : Table Row = PLC HMI.partCall.current[10], 100 ms

text list "Station Selection Single": 0 'Select a Station to View'; 1 'Station Assignments'

screen "1 PART CALL" 1366x768
   on GenerateScreen: SetTag("HMI_screenNumber", 1)
   Rectangle "Nav Panel 02" at 682,700 size 684x68
      Appearance <- "HMI_screenNumber"
   Rectangle "Nav Panel 01" at 0,700 size 685x68
      Appearance <- "HMI_screenNumber"
   Rectangle "Nav Panel 03 Top Border Hide" at 685,700 size 678x3
      Visibility <- "HMI_screenNumber"
   Rectangle "Nav Panel 01 Top Border Hide" at 3,700 size 679x3
      Visibility <- "HMI_screenNumber"
   Button "Settings Screen" at 683,700 size 683x68; TextOff 'SETTINGS'; Authorization "User administration"
      on Release: ActivateScreen("2 SETTINGS", 0)
   Button "Part Call Screen" at 0,700 size 683x68; TextOff 'PART CALL'
      on Release: ActivateScreen("1 PART CALL", 0)
   TextField "Header Line" at 32,32 size 216x53; Text 'LINE'
   TextField "Header Drop Zone" at 238,32 size 236x53; Text 'DROP ZONE'
   TextField "Header Part Number" at 474,32 size 648x53; Text 'PART NUMBER'
   TextField "Header Time" at 1112,32 size 222x53; Text 'TIME'
   ScreenModuleView "TableRow00" at 27,90 size 1312x52; ScreenModuleType ""
      Guid_{11997190-27688} <- "HMI_partCall_current{0}"
   ScreenModuleView "TableRow01" at 27,142 size 1312x52; ScreenModuleType ""
      Guid_{11997190-27688} <- "HMI_partCall_current{1}"
   ScreenModuleView "TableRow02" at 27,194 size 1312x52; ScreenModuleType ""
      Guid_{11997190-27688} <- "HMI_partCall_current{2}"
   ScreenModuleView "TableRow03" at 27,246 size 1312x52; ScreenModuleType ""
      Guid_{11997190-27688} <- "HMI_partCall_current{3}"
   ScreenModuleView "TableRow04" at 27,298 size 1312x52; ScreenModuleType ""
      Guid_{11997190-27688} <- "HMI_partCall_current{4}"
   ScreenModuleView "TableRow05" at 27,350 size 1312x52; ScreenModuleType ""
      Guid_{11997190-27688} <- "HMI_partCall_current{5}"
   ScreenModuleView "TableRow06" at 27,402 size 1312x52; ScreenModuleType ""
      Guid_{11997190-27688} <- "HMI_partCall_current{6}"
   ScreenModuleView "TableRow07" at 27,454 size 1312x52; ScreenModuleType ""
      Guid_{11997190-27688} <- "HMI_partCall_current{7}"
   ScreenModuleView "TableRow08" at 27,506 size 1312x52; ScreenModuleType ""
      Guid_{11997190-27688} <- "HMI_partCall_current{8}"
   ScreenModuleView "TableRow09" at 27,558 size 1312x52; ScreenModuleType ""
      Guid_{11997190-27688} <- "HMI_partCall_current{9}"
   ScreenModuleView "TableRow10" at 27,610 size 1312x52; ScreenModuleType ""
      Guid_{11997190-27688} <- "HMI_partCall_current{10}"

screen "2 SETTINGS" 1366x768
   on GenerateScreen: SetTag("HMI_screenNumber", 2)
   Rectangle "Nav Panel 01" at 0,700 size 685x68
      Appearance <- "HMI_screenNumber"
   Rectangle "Nav Panel 02" at 682,700 size 684x68
      Appearance <- "HMI_screenNumber"
   Rectangle "Station Assignment Table BG Full" at 793,40 size 533x630
      Visibility <- "selCount"
   Button "Part Call Screen" at 0,700 size 683x68; TextOff 'PART CALL'
      on Release: ActivateScreen("1 PART CALL", 0)
   Button "Settings Screen" at 683,700 size 683x68; TextOff 'SETTINGS'
      on Release: ActivateScreen("2 SETTINGS", 0)
   IOField "I/O field_1" at 50,100 size 414x50; FormatPattern ????????????????????
      ObjectEnable <- "enable"
      Appearance <- "enable"
      ProcessValue <- "value"
   IOField "I/O field_2" at 494,100 size 137x50; FormatPattern ?????
      Appearance <- "enable"
      ObjectEnable <- "enable"
      ProcessValue <- "value"
   IOField "I/O field_3" at 636,100 size 137x50; FormatPattern ?????
      ObjectEnable <- "enable"
      Appearance <- "enable"
      ProcessValue <- "value"
   Button "Assign All Stations" at 120,190 size 274x45; TextOff 'Select Stations'
      on Press: function_b14e0dd5("act", 0)
      Appearance <- "enable"
      ObjectEnable <- "enable"
   Button "Station 1 Select" at 50,240 size 205x65; TextOff 'Text'
      Appearance <- "[0]"
      on Press: function_b14e0dd5("select", 0)
   Button "Station 2 Select" at 261,240 size 203x65; TextOff 'Text'
      Appearance <- "[1]"
      on Press: function_b14e0dd5("select", 0)
   Button "Station 3 Select" at 50,311 size 205x65; TextOff 'Text'
      Appearance <- "[2]"
      on Press: function_b14e0dd5("select", 0)
   Button "Station 4 Select" at 261,311 size 203x65; TextOff 'Text'
      Appearance <- "[3]"
      on Press: function_b14e0dd5("select", 0)
   Button "Station 5 Select" at 50,382 size 205x65; TextOff 'Text'
      Appearance <- "[4]"
      on Press: function_b14e0dd5("select", 0)
   Button "Station 6 Select" at 261,382 size 203x65; TextOff 'Text'
      Appearance <- "[5]"
      on Press: function_b14e0dd5("select", 0)
   Button "Station 7 Select" at 50,453 size 205x65; TextOff 'Text'
      Appearance <- "[6]"
      on Press: function_b14e0dd5("select", 0)
   Button "Station 8 Select" at 261,453 size 203x65; TextOff 'Text'
      Appearance <- "[7]"
      on Press: function_b14e0dd5("select", 0)
   Button "Station 9 Select" at 50,524 size 205x65; TextOff 'Text'
      Appearance <- "[8]"
      on Press: function_b14e0dd5("select", 0)
   Button "Station 10 Select" at 261,524 size 203x65; TextOff 'Text'
      Appearance <- "[9]"
      on Press: function_b14e0dd5("select", 0)
   Button "Station 11 Select" at 50,595 size 205x65; TextOff 'Text'
      Appearance <- "[10]"
      on Press: function_b14e0dd5("select", 0)
   Button "Enable Part Entry" at 50,50 size 414x45; TextOff 'Enter Part Number'
      on Press: function_b14e0dd5("enter", 0)
      Appearance <- "enable"
      ObjectEnable <- "enable"
   Button "Enable Set Timer" at 494,50 size 137x45; TextOff 'Timer'
      on Press: function_b14e0dd5("setTimer", 0)
      ObjectEnable <- "enable"
      Appearance <- "enable"
   Button "Enable Set Timer_1" at 636,50 size 137x45; TextOff 'Critical'
      on Press: function_b14e0dd5("setTimer", 0)
      ObjectEnable <- "enable"
      Appearance <- "enable"
   Button "Station 11 Select_1" at 261,595 size 205x65; TextOff 'Text'
      Appearance <- "[11]"
      on Press: function_b14e0dd5("select", 0)
   TextField "Current Station Single" at 803,50 size 513x45; Text 'Text'
      Visibility <- "HMI_screenNumber"
   Button "Previous Station" at 803,50 size 65x45; TextOff 'Text'; PictureOff "Graphic_1"
      on Press: function_b14e0dd5("act", 0)
      Visibility <- "selCount"
      Appearance <- "ani"
   Button "Next Station" at 1251,50 size 65x45; TextOff 'Text'; PictureOff "Graphic_2"
      on Press: function_b14e0dd5("act", 0)
      Visibility <- "selCount"
      Appearance <- "act"
   TextField "Current Station Multi" at 873,50 size 373x45; Text 'Station Assignments'
      Visibility <- "selCount"
   Button "Previous Station_1" at 50,190 size 65x45; TextOff 'Text'; PictureOff "Graphic_1"
      on Press: function_b14e0dd5("act", 0)
      Appearance <- "ani"
      Visibility <- "enable"
      ObjectEnable <- "enable"
   Button "Next Station_1" at 399,190 size 65x45; TextOff 'Text'; PictureOff "Graphic_2"
      on Press: function_b14e0dd5("act", 0)
      Appearance <- "ani"
      Visibility <- "enable"
      ObjectEnable <- "enable"
   Rectangle "Station Assignment Table BG Mini" at 793,40 size 533x65
      Visibility <- "selCount"
   Rectangle "Nav Panel 01 Top Border Hide" at 3,700 size 679x3
      Visibility <- "HMI_screenNumber"
   Rectangle "Nav Panel 03 Top Border Hide" at 685,700 size 678x3
      Visibility <- "HMI_screenNumber"
   Button "Select All Buttons" at 493,190 size 284x45; TextOff 'Assign to Buttons'
      on Press: function_b14e0dd5("act", 0)
      Appearance <- "ani"
      ObjectEnable <- "enable"
   GraphicView "KP8 Image" at 496,247 size 275x412; Picture "kp8 image"
   Button "KP8 7" at 557,303 size 68x66; TextOff '1'
      on Press: function_b14e0dd5("select", 0)
      Appearance <- "animation"
   Button "KP8 3" at 641,303 size 68x66; TextOff '2'
      on Press: function_b14e0dd5("select", 0)
      Appearance <- "animation"
   Button "KP8 6" at 557,379 size 68x66; TextOff '3'
      Appearance <- "animation"
      on Press: function_b14e0dd5("select", 0)
   Button "KP8 2" at 641,379 size 68x66; TextOff '4'
      Appearance <- "animation"
      on Press: function_b14e0dd5("select", 0)
   Button "KP8 5" at 557,456 size 68x66; TextOff '5'
      Appearance <- "animation"
      on Press: function_b14e0dd5("select", 0)
   Button "KP8 1" at 641,456 size 68x66; TextOff '6'
      Appearance <- "animation"
      on Press: function_b14e0dd5("select", 0)
   Button "KP8 4" at 557,532 size 68x66; TextOff 'NOT USED'
      on Release: StopRuntime(0)
   Button "KP8 0" at 641,532 size 68x66; TextOff 'NOT USED'
   TextField "Button 6 Label" at 803,586 size 75x74; Text '6'
      Visibility <- "selCount"
   TextField "Button 6 Timer" at 866,586 size 107x37; Text 'Text'
      Visibility <- "selCount"
   TextField "Button 6 Part Number" at 968,586 size 348x74; Text 'Text'
      Visibility <- "selCount"
   TextField "Button 5 Label" at 803,507 size 75x74; Text '5'
      Visibility <- "selCount"
   TextField "Button 5 Timer" at 866,507 size 107x37; Text 'Text'
      Visibility <- "selCount"
   TextField "Button 5 Part Number" at 968,507 size 348x74; Text 'Text'
      Visibility <- "selCount"
   TextField "Button 4 Label" at 803,428 size 75x74; Text '4'
      Visibility <- "selCount"
   TextField "Button 4 Timer" at 866,428 size 107x37; Text 'Text'
      Visibility <- "selCount"
   TextField "Button 4 Part Number" at 968,428 size 348x74; Text 'Text'
      Visibility <- "selCount"
   TextField "Button 3 Label" at 803,349 size 75x74; Text '3'
      Visibility <- "selCount"
   TextField "Button 3 Timer" at 866,349 size 107x37; Text 'Text'
      Visibility <- "selCount"
   TextField "Button 3 Part Number" at 968,349 size 348x74; Text 'Text'
      Visibility <- "selCount"
   TextField "Button 2 Label" at 803,270 size 75x74; Text '2'
      Visibility <- "selCount"
   TextField "Button 2 Timer" at 866,270 size 107x37; Text 'Text'
      Visibility <- "selCount"
   TextField "Button 2 Part Number" at 968,270 size 348x74; Text 'Text'
      Visibility <- "selCount"
   TextField "Button 1 Label" at 803,191 size 75x74; Text '1'
      Visibility <- "selCount"
   TextField "Button 1 Timer" at 866,191 size 107x37; Text 'Text'
      Visibility <- "selCount"
   TextField "Button 1 Part Number" at 968,191 size 348x74; Text 'Text'
      Visibility <- "selCount"
   TextField "Button Column Header" at 803,146 size 75x40; Text 'Btn'
      Visibility <- "selCount"
   TextField "Timer Column Header" at 866,146 size 107x40; Text 'Times'
      Visibility <- "selCount"
   TextField "Part Number Column Header" at 968,146 size 348x40; Text 'Part Number'
      Visibility <- "selCount"
   TextField "Button 1 Timer_1" at 866,228 size 107x37; Text 'Text'
      Visibility <- "selCount"
   TextField "Button 1 Timer_2" at 866,307 size 107x37; Text 'Text'
      Visibility <- "selCount"
   TextField "Button 1 Timer_3" at 866,386 size 107x37; Text 'Text'
      Visibility <- "selCount"
   TextField "Button 1 Timer_4" at 866,465 size 107x37; Text 'Text'
      Visibility <- "selCount"
   TextField "Button 1 Timer_5" at 866,544 size 107x37; Text 'Text'
      Visibility <- "selCount"
   TextField "Button 1 Timer_6" at 866,623 size 107x37; Text 'Text'
      Visibility <- "selCount"
   TextField "Drop Zone Label" at 1076,101 size 240x40; Text 'Drop Zone:'
      Visibility <- "selCount"
   TextField "Line Label" at 803,101 size 267x40; Text 'Line:'
      Visibility <- "selCount"
   TextField "Hide Line and Drop Zone Multi" at 803,101 size 513x40; Text 'select single station for Line and Drop Zone'
      Visibility <- "selCount"
   IOField "Line" at 889,101 size 181x40; FormatPattern ?????????
      Visibility <- "selCount"
      ProcessValue <- "lineValue"
   IOField "Drop Zone Entry" at 1247,101 size 69x40; FormatPattern 999
      Visibility <- "selCount"
      ProcessValue <- "dzValue"

screen "3 BARCODE" 1366x768
   on GenerateScreen: SetTag("HMI_screenNumber", 3)
   Rectangle "Nav Panel 02" at 682,700 size 684x68
      Appearance <- "HMI_screenNumber"
   Rectangle "Nav Panel 01" at 0,700 size 685x68
      Appearance <- "HMI_screenNumber"
   Rectangle "Nav Panel 03 Top Border Hide" at 685,700 size 678x3
      Visibility <- "HMI_screenNumber"
   Rectangle "Nav Panel 01 Top Border Hide" at 3,700 size 679x3
      Visibility <- "HMI_screenNumber"
   Button "Settings Screen" at 683,700 size 683x68; TextOff 'SETTINGS'; Authorization "User administration"
      on Release: ActivateScreen("2 SETTINGS", 0)
   Button "Part Call Screen" at 0,700 size 683x68; TextOff 'PART CALL'
      on Release: ActivateScreen("1 PART CALL", 0)
   Button "btCancel" at 685,431 size 649x68; TextOff 'CANCEL'
      on Release: ActivateScreen("1 PART CALL", 0)
   Button "btPartOrdered" at 32,431 size 648x68; TextOff 'ORDERED'
      on Release: SetBit("ordered"); ActivateScreen("1 PART CALL", 0)
   TextField "tfBarcodeDisplay" at 32,220 size 1302x206; Text 'Text'
   TextField "tfPartNumberDisplay" at 32,160 size 1302x53; Text 'BARCODE FOR PART NUMBER'
*)

(* ===== HMI "HMI_RT_2" =====
connection "HMI_Connection_3": ETHERNET, S7_1500_OMS

HMI tags "Default tag table"
   "Clock_0.5Hz" : Bool = PLC "Clock_0.5Hz" AT %M0.7, 100 ms
   "HMI_Drop Zone" : Array [0..65] of WString[20] = PLC "EMP IDB".HMI."Part Call"."Drop Zone" AT %DB1.DBX0.0, 100 ms
   "HMI_Flash Request" : Array [0..65] of USInt = PLC "EMP IDB".HMI."Part Call"."Flash Request" AT %DB1.DBX0.0, 100 ms
   "HMI_Line" : Array [0..65] of WString[20] = PLC "EMP IDB".HMI."Part Call".Line AT %DB1.DBB0, 100 ms
   "HMI_Number of Rows" : USInt = PLC "EMP IDB".HMI."Part Call"."Number of Rows" AT %DB1.DBW0, 100 ms
   "HMI_Part Numbers" : Array [0..65] of WString[20] = PLC "EMP IDB".HMI."Part Call"."Part Numbers" AT %DB1.DBX0.0, 100 ms
   "HMI_Time" : Array [0..65] of WString[10] = PLC "EMP IDB".HMI."Part Call".Time AT %DB1.DBX0.0, 100 ms

screen "1 PART CALL" 1024x768
   Rectangle "Connection Status" at 1,196 size 894x1
      Appearance <- "Clock_0.5Hz"
   TextField "C0R0 Line" at 6,9 size 110x28; Text 'Text'
      Visibility <- "HMI_Number of Rows"
      Appearance <- "[0]"
   TextField "C0R0 Drop Zone" at 111,9 size 42x28; Text 'Text'
      Visibility <- "HMI_Number of Rows"
      Appearance <- "[0]"
   TextField "C0R0 Part Number" at 153,9 size 209x28; Text 'Text'
      Visibility <- "HMI_Number of Rows"
      Appearance <- "[0]"
   TextField "C0R0 Time" at 360,9 size 86x28; Text 'Text'
      Visibility <- "HMI_Number of Rows"
      Appearance <- "[0]"
   TextField "C0R1 Line" at 6,39 size 110x28; Text 'Text'
      Visibility <- "HMI_Number of Rows"
      Appearance <- "[1]"
   TextField "C0R1 Drop Zone" at 111,39 size 42x28; Text 'Text'
      Visibility <- "HMI_Number of Rows"
      Appearance <- "[1]"
   TextField "C0R1 Part Number" at 153,39 size 209x28; Text 'Text'
      Visibility <- "HMI_Number of Rows"
      Appearance <- "[1]"
   TextField "C0R1 Time" at 360,39 size 86x28; Text 'Text'
      Visibility <- "HMI_Number of Rows"
      Appearance <- "[1]"
   TextField "C0R2 Line" at 6,69 size 110x28; Text 'Text'
      Visibility <- "HMI_Number of Rows"
      Appearance <- "[2]"
   TextField "C0R2 Drop Zone" at 111,69 size 42x28; Text 'Text'
      Visibility <- "HMI_Number of Rows"
      Appearance <- "[2]"
   TextField "C0R2 Part Number" at 153,69 size 209x28; Text 'Text'
      Visibility <- "HMI_Number of Rows"
      Appearance <- "[2]"
   TextField "C0R2 Time" at 360,69 size 86x28; Text 'Text'
      Visibility <- "HMI_Number of Rows"
      Appearance <- "[2]"
   TextField "C0R3 Line" at 6,99 size 110x28; Text 'Text'
      Visibility <- "HMI_Number of Rows"
      Appearance <- "[3]"
   TextField "C0R3 Drop Zone" at 111,99 size 42x28; Text 'Text'
      Visibility <- "HMI_Number of Rows"
      Appearance <- "[3]"
   TextField "C0R3 Part Number" at 153,99 size 209x28; Text 'Text'
      Visibility <- "HMI_Number of Rows"
      Appearance <- "[3]"
   TextField "C0R3 Time" at 360,99 size 86x28; Text 'Text'
      Visibility <- "HMI_Number of Rows"
      Appearance <- "[3]"
   TextField "C0R4 Line" at 6,128 size 110x28; Text 'Text'
      Visibility <- "HMI_Number of Rows"
      Appearance <- "[4]"
   TextField "C0R4 Drop Zone" at 111,128 size 42x28; Text 'Text'
      Visibility <- "HMI_Number of Rows"
      Appearance <- "[4]"
   TextField "C0R4 Part Number" at 153,128 size 209x28; Text 'Text'
      Visibility <- "HMI_Number of Rows"
      Appearance <- "[4]"
   TextField "C0R4 Time" at 360,128 size 86x28; Text 'Text'
      Visibility <- "HMI_Number of Rows"
      Appearance <- "[4]"
   TextField "C0R5 Line" at 6,158 size 110x28; Text 'Text'
      Visibility <- "HMI_Number of Rows"
      Appearance <- "[5]"
   TextField "C0R5 Drop Zone" at 111,158 size 42x28; Text 'Text'
      Visibility <- "HMI_Number of Rows"
      Appearance <- "[5]"
   TextField "C0R5 Part Number" at 153,158 size 209x28; Text 'Text'
      Visibility <- "HMI_Number of Rows"
      Appearance <- "[5]"
   TextField "C0R5 Time" at 360,158 size 86x28; Text 'Text'
      Visibility <- "HMI_Number of Rows"
      Appearance <- "[5]"
   TextField "C1R0 Line" at 455,9 size 110x28; Text 'Text'
      Visibility <- "HMI_Number of Rows"
      Appearance <- "[6]"
   TextField "C1R0 Drop Zone" at 560,9 size 42x28; Text 'Text'
      Visibility <- "HMI_Number of Rows"
      Appearance <- "[6]"
   TextField "C1R0 Part Number" at 602,9 size 209x28; Text 'Text'
      Visibility <- "HMI_Number of Rows"
      Appearance <- "[6]"
   TextField "C1R0 Time" at 809,9 size 84x28; Text 'Text'
      Visibility <- "HMI_Number of Rows"
      Appearance <- "[6]"
   TextField "Row 1 Line_1" at 455,39 size 110x28; Text 'Text'
      Visibility <- "HMI_Number of Rows"
      Appearance <- "[7]"
   TextField "Row 1 Drop Zone_1" at 560,39 size 42x28; Text 'Text'
      Visibility <- "HMI_Number of Rows"
      Appearance <- "[7]"
   TextField "Row 1 Part Number_1" at 602,39 size 209x28; Text 'Text'
      Visibility <- "HMI_Number of Rows"
      Appearance <- "[7]"
   TextField "Row 1 Time_1" at 809,39 size 84x28; Text 'Text'
      Visibility <- "HMI_Number of Rows"
      Appearance <- "[7]"
   TextField "Row 2 Line_1" at 455,69 size 110x28; Text 'Text'
      Visibility <- "HMI_Number of Rows"
      Appearance <- "[8]"
   TextField "Row 2 Drop Zone_1" at 560,69 size 42x28; Text 'Text'
      Visibility <- "HMI_Number of Rows"
      Appearance <- "[8]"
   TextField "Row 2 Part Number_1" at 602,69 size 209x28; Text 'Text'
      Visibility <- "HMI_Number of Rows"
      Appearance <- "[8]"
   TextField "Row 2 Time_1" at 809,69 size 84x28; Text 'Text'
      Visibility <- "HMI_Number of Rows"
      Appearance <- "[8]"
   TextField "Row 3 Line_1" at 455,99 size 110x28; Text 'Text'
      Visibility <- "HMI_Number of Rows"
      Appearance <- "[9]"
   TextField "Row 3 Drop Zone_1" at 560,99 size 42x28; Text 'Text'
      Visibility <- "HMI_Number of Rows"
      Appearance <- "[9]"
   TextField "Row 3 Part Number_1" at 602,99 size 209x28; Text 'Text'
      Visibility <- "HMI_Number of Rows"
      Appearance <- "[9]"
   TextField "Row 3 Time_1" at 809,99 size 84x28; Text 'Text'
      Visibility <- "HMI_Number of Rows"
      Appearance <- "[9]"
   TextField "Row 4 Line_1" at 455,128 size 110x28; Text 'Text'
      Visibility <- "HMI_Number of Rows"
      Appearance <- "[10]"
   TextField "Row 4 Drop Zone_1" at 560,128 size 42x28; Text 'Text'
      Visibility <- "HMI_Number of Rows"
      Appearance <- "[10]"
   TextField "Row 4 Part Number_1" at 602,128 size 209x28; Text 'Text'
      Visibility <- "HMI_Number of Rows"
      Appearance <- "[10]"
   TextField "Row 4 Time_1" at 809,128 size 84x28; Text 'Text'
      Visibility <- "HMI_Number of Rows"
      Appearance <- "[10]"
   TextField "Row 5 Line_1" at 455,158 size 110x28; Text 'Text'
      Visibility <- "HMI_Number of Rows"
      Appearance <- "[11]"
   TextField "Row 5 Drop Zone_1" at 560,158 size 42x28; Text 'Text'
      Visibility <- "HMI_Number of Rows"
      Appearance <- "[11]"
   TextField "Row 5 Part Number_1" at 602,158 size 209x28; Text 'Text'
      Visibility <- "HMI_Number of Rows"
      Appearance <- "[11]"
   TextField "Row 5 Time_1" at 809,158 size 84x28; Text 'Text'
      Visibility <- "HMI_Number of Rows"
      Appearance <- "[11]"
*)

(* ===== HMI "HMI_RT_1" =====
system functions are stored by id; their names below are inferred from use

ScreenModuleEditorView "Table Row" 1312x52
   TextField "tfLine" at 5,1 size 216x48; Text 'Text'
      Visibility <- "interface.tfLine.visibility"
      Appearance <- "interface.tfLine.animator"
   TextField "tfTime" at 1085,1 size 222x48; Text 'Text'
      Appearance <- "interface.tfTime.animator"
      Visibility <- "interface.tfTime.visibility"
   TextField "tfDropZone" at 211,1 size 236x48; Text 'Text'
      Appearance <- "interface.tfDropZone.animator"
      Visibility <- "interface.tfDropZone.visibility"
   TextField "tfPartNumber" at 445,1 size 650x48; Text 'Text'
      Appearance <- "interface.tfPartNumber.animator"
      Visibility <- "interface.tfPartNumber.visibility"
   Button "pbSelect" at 0,0 size 1312x52; TextOff 'Text'
      Visibility <- "interface.pbSelection.visibility"
      on Press: SetBit("interface.pbSelection.request")
      on Release: ResetBit("interface.pbSelection.request")
   Rectangle "rtBackground" at 0,0 size 1312x52
      Visibility <- "interface.rtBackground.visibility"
*)

(* ===== HMI "HMI_RT_1" =====
system functions are stored by id; their names below are inferred from use

ScreenModuleEditorView "Table Row" 1312x52
   TextField "tfLine" at 5,1 size 216x48; Text 'Text'
      Visibility <- "interface.tfLine.visibility"
      Appearance <- "interface.tfLine.animator"
   TextField "tfTime" at 1085,1 size 222x48; Text 'Text'
      Visibility <- "interface.tfTime.visibility"
      Appearance <- "interface.tfTime.animator"
   TextField "tfDropZone" at 211,1 size 236x48; Text 'Text'
      Visibility <- "interface.tfDropZone.visibility"
      Appearance <- "interface.tfDropZone.animator"
   TextField "tfPartNumber" at 445,1 size 650x48; Text 'Text'
      Visibility <- "interface.tfPartNumber.visibility"
      Appearance <- "interface.tfPartNumber.animator"
   Button "pbSelect" at 0,0 size 1312x52; TextOff 'Text'
      on Release: ResetBit("interface.pbSelection.request")
      on Press: SetBit("interface.pbSelection.request")
      Visibility <- "interface.pbSelection.visibility"
   Rectangle "rtBackground" at 0,0 size 1312x52
      Visibility <- "interface.rtBackground.visibility"
*)